(* CODESYS project Test02.project

Project tree, tasks and I/O mapping:
  Device : Elmo Platinum Maestro, Elmo Motion Control, version 1.0.0.2
    application Application
      libraries: Standard, * (System)
      task MainTask (cyclic, interval t#20ms, priority 1) calls PLC_PRG
      task VISU_TASK (cyclic, interval 100 ms, priority 31) calls VisuElems.Visu_Prg
      program PLC_PRG [ST]
      visualisation VisuTest01
      01_Enumerator/
        data type eStatus
      Structure/
        data type stBall
    Elmo_Master_Device : Elmo Master Device, Elmo, version 1.0.0.2
  libraries: VisuSymbols, 3.5.10.0 (System)
  text list GlobalTextList
*)

// Device/Application/01_Enumerator/eStatus
{attribute 'qualified_only'}
{attribute 'strict'}
TYPE eStatus :
(
	//enum_member := 0
	xPositive := 0,
	yNegative := 100,
	xNegative := 200,
	yPositive := 300
);
END_TYPE

// Device/Application/Structure/stBall
TYPE stBall :
STRUCT
	iMove_x : INT;
	iMove_y : INT;
	dwColor : DWORD;
	sStatus: STRING;
END_STRUCT
END_TYPE

// Device/Application/PLC_PRG
PROGRAM PLC_PRG
VAR
	xBtn : BOOL;
	xLight : BOOL;
	sIndicator : STRING;
	iCnt : INT;
	rCnt : REAL;
	xTemp : BOOL := TRUE;
	iMove_x : INT;
	iMove_y : INT;
	iMove_z : INT;
	stBallA: stBall;
END_VAR

xLight := xBtn;

IF xLight THEN
	sIndicator := 'ON';
ELSE
	sIndicator := 'OFF';
END_IF

//iCnt := iCnt + 1;
rCnt := rCnt + 0.1; 


IF iCnt <= 1000 AND xTemp THEN
//IF iCnt <= 1000 THEN
	iCnt := iCnt + 1;
ELSE
	(*
	FOR iCnt:=iCnt TO 0 BY -1 DO
		   iCnt := iCnt - 1;
	END_FOR
	*)
	
	xTemp := FALSE;
	iCnt := iCnt - 1;
	IF iCnt = 0 THEN
		xTemp := TRUE;
	END_IF
	
	
END_IF

//iMove_x := 0;
//iMove_y := 0;

CASE iMove_z OF
	eStatus.xPositive:
	   //iMove_x:= iMove_x + 1;
	   stBallA.iMove_x := stBallA.iMove_x + 1;
	   stBallA.dwColor := 16#FFFF0000;
	   stBallA.sStatus := 'Moving right';
	   IF stBallA.iMove_x = 100 THEN
	       iMove_z:= eStatus.yNegative;
	   END_IF
	   (*
	   WHILE iMove_x < 100 DO
	      iMove_x := iMove_x + 1;
       END_WHILE
	   *)
	   
	   //iMove_x:= iMove_x + 1;
	   
	eStatus.yNegative:
	   //iMove_x:= 20;
	   stBallA.iMove_y:= stBallA.iMove_y + 1;
	   stBallA.dwColor := 16#FFFFFF00;
	   stBallA.sStatus := 'Moving down';
	   IF stBallA.iMove_y = 100 THEN
	       iMove_z:= eStatus.xNegative;
	   END_IF
	eStatus.xNegative:
	   stBallA.iMove_x := stBallA.iMove_x - 1;
	   stBallA.dwColor := 16#FF00FF00;
	   stBallA.sStatus := 'Moving left';
	   IF stBallA.iMove_x = 0 THEN
	       iMove_z:= eStatus.yPositive;
	   END_IF
	   //WHILE iMove_x >  -3 DO
	     // iMove_x := iMove_x - 2;
       //END_WHILE
	   
	eStatus.yPositive:
	  //WHILE iMove_y >  0 DO
	  stBallA.iMove_y := stBallA.iMove_y - 1;
	  stBallA.dwColor := 16#88888888;
	  stBallA.sStatus := 'Moving up';
	   IF stBallA.iMove_y = 0 THEN
	       iMove_z:= eStatus.xPositive;
	   END_IF
	   //iMove_y := iMove_y - 100;
       //END_WHILE
	   //iMove_x := 0;
	   (*
	   WHILE iMove_y < 100 DO
	      iMove_y := iMove_y + 1;
       END_WHILE
	   WHILE iMove_x > 0 DO
	      iMove_x := iMove_y - 1;
       END_WHILE
	   WHILE iMove_y > 100 DO
	      iMove_y := iMove_y - 1;
       END_WHILE
	   *)
	   (*
	   IF iMove_y = 100 THEN
		   iMove_x:= iMove_x - 1;
		   IF iMove_x = 0 THEN
			   iMove_y:= iMove_y - 1;
		   END_IF
	   END_IF
	   *)
	(*
	20:
	   iMove_x:= 30;
	30:
	   iMove_x:= 40;
	   *)
	//99:
	  //iMove_x:= 1;
	//ELSE
		//iMove_y:= 0;
		//iMove_x:= 0;
		
END_CASE

(*
CASE iMove_y OF
	100:
	  iMove_x:= iMove_x + 1;
	1:
	  iMove_x:= iMove_x - 1;
	  *)
	
//END_CASE

END_PROGRAM

// Device/Application/VisuTest01
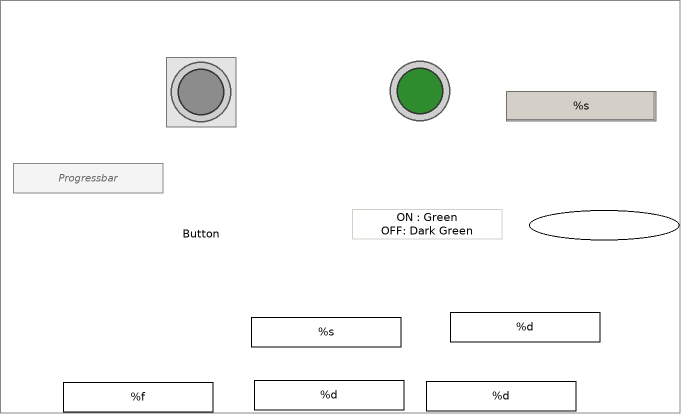
VISUALIZATION VisuTest01  // 681x414
    Lamp1 (385,56 70x70), variable: PLC_PRG.xLight, style: Lamp-Lamp1-Green
    PushSwitch (166,57 70x70), variable: PLC_PRG.xBtn, behaviour: TOGGLE, style: Switch-PushSwitch-Gray
    Label (126,219 150x30), "Button"
    Textfield (352,209 150x30), "ON : Green OFF: Dark Green"
    Rectangle (251,317 150x30), "%s", text variable: PLC_PRG.sIndicator
    Rectangle (450,312 150x30), "%d", text variable: PLC_PRG.iCnt
    Rectangle (63,382 150x30), "%f", text variable: PLC_PRG.rCnt
    Button (506,91 150x30), "%s", text variable: PLC_PRG.sIndicator
        toggle PLC_PRG.xBtn
    Progressbar (13,163 150x30), variable: PLC_PRG.iCnt
    Ellipse (529,210 150x30), colour variable: PLC_PRG.stBallA.dwColor
        p3560616238: PLC_PRG.stBallA.iMove_x
        p2738717112: PLC_PRG.stBallA.iMove_y
    Rectangle (254,380 150x30), "%d", text variable: PLC_PRG.stBallA.iMove_x
    Rectangle (426,381 150x30), "%d", text variable: PLC_PRG.stBallA.iMove_y
END_VISUALIZATION
